Universal Robots URScript: test.script

def unnamed():
  set_tcp(p[-0.12,-0.038,0.18,0.0,0.0,0.0])
  set_payload(1.75, [-0.11671, -0.042, 0.015])
  set_tool_voltage(0)
  set_gravity([0.0, -1.2026031567627009E-15, -9.82])
  set_standard_analog_input_domain(0, 1)
  set_standard_analog_input_domain(1, 1)
  set_tool_analog_input_domain(0, 1)
  set_tool_analog_input_domain(1, 1)
  set_analog_outputdomain(0, 0)
  set_analog_outputdomain(1, 0)
  set_input_actions_to_default()
  set_runstate_gp_boolean_output_to_value(74, 3)
  step_count_ce4ce9db_3ae8_46aa_94b7_30826356951c = 0.0
  thread Step_Counter_Thread_22e32eef_2b87_4dae_bee3_4c02b1791a95():
    while (True):
      step_count_ce4ce9db_3ae8_46aa_94b7_30826356951c = step_count_ce4ce9db_3ae8_46aa_94b7_30826356951c + 1.0
      sync()
    end
  end
  run Step_Counter_Thread_22e32eef_2b87_4dae_bee3_4c02b1791a95()
  set_safety_mode_transition_hardness(1)
  global Base=p[0.0,0.0,0.0,0.0,0.0,0.0]
  global stack_a=p[-0.4452193668035932,-0.5335582242141723,1.2187665551547486,-1.4775023178422264,0.6206358915374167,-0.5973276910217602]
  global stack_b=p[-0.5217422958491581,-0.5417780095732599,1.2153549374776276,-1.4758179672679694,0.5899140330979058,-0.5966029981778683]
  while (True):
    $ 1 "Robot Program"
    $ 2 "var_1≔p[-0.2,0.2,0.2,0,3.1415,0]"
    global var_1=p[-0.2,0.2,0.2,0,3.1415,0]
    $ 3 "MoveJ"
    $ 4 "var_1" "breakAfter"
    movej(var_1, a=1.3962634015954636, v=1.0471975511965976)
  end
end
